// TIA Portal V17 export
// export: Created 2024-08-29T18:23:47.92153Z, ExportSetting WithDefaults, DisplayName Totally Integrated Automation Portal, DisplayVersion V17 Update 7, DisplayName TIA Portal Openness, DisplayVersion V17 Update 7, DisplayName TIA Portal Version Control Interface, DisplayVersion V17, DisplayName SINAMICS Startdrive Advanced, DisplayVersion V17 SP2, DisplayName SINAMICS Startdrive G110M, G120, G120C, G120D, G120P, G115D, DisplayVersion V17 SP2, DisplayName SINAMICS Startdrive G130, G150, S120, S150, SINAMICS MV, S210, DisplayVersion V17 SP2, DisplayName STEP 7 Professional, DisplayVersion V17 Update 7, DisplayName STEP 7 Safety, DisplayVersion V17 Update 6, DisplayName WinCC Advanced / Unified PC, DisplayVersion V17 Update 7
DATA_BLOCK "DB_SEND_IJCORE"   // DB1005
{ S7_Optimized_Access := 'FALSE' }
VERSION : 0.1
// stored: AutoNumber false, DBAccessibleFromOPCUA true, DBAccessibleFromWebserver true, IsOnlyStoredInLoadMemory false, IsWriteProtectedInAS false
   VAR
      Awake_DW : Word := 16#0000;
      Awake_SW : Int := 1;
      SW_Message : Array[1..300] of Word;
      Message : Array[1..50] of Struct
         Content : Array[1..80] of Byte;
      END_STRUCT;
   END_VAR
BEGIN
   SW_Message[1..8] := 16#FFFF;
   SW_Message[9..300] := 16#0000;
   Message[1].Content[1..80] := 16#00;
   Message[2].Content[1..80] := 16#00;
   Message[3].Content[1..80] := 16#00;
   Message[4].Content[1..80] := 16#00;
   Message[5].Content[1..80] := 16#00;
   Message[6].Content[1..80] := 16#00;
   Message[7].Content[1..80] := 16#00;
   Message[8].Content[1..80] := 16#00;
   Message[9].Content[1..80] := 16#00;
   Message[10].Content[1..80] := 16#00;
   Message[11].Content[1..80] := 16#00;
   Message[12].Content[1..80] := 16#00;
   Message[13].Content[1..80] := 16#00;
   Message[14].Content[1..80] := 16#00;
   Message[15].Content[1..80] := 16#00;
   Message[16].Content[1..80] := 16#00;
   Message[17].Content[1..80] := 16#00;
   Message[18].Content[1..80] := 16#00;
   Message[19].Content[1..80] := 16#00;
   Message[20].Content[1..80] := 16#00;
   Message[21].Content[1..80] := 16#00;
   Message[22].Content[1..80] := 16#00;
   Message[23].Content[1..80] := 16#00;
   Message[24].Content[1..80] := 16#00;
   Message[25].Content[1..80] := 16#00;
   Message[26].Content[1..80] := 16#00;
   Message[27].Content[1..80] := 16#00;
   Message[28].Content[1..80] := 16#00;
   Message[29].Content[1..80] := 16#00;
   Message[30].Content[1..80] := 16#00;
   Message[31].Content[1..80] := 16#00;
   Message[32].Content[1..80] := 16#00;
   Message[33].Content[1..80] := 16#00;
   Message[34].Content[1..80] := 16#00;
   Message[35].Content[1..80] := 16#00;
   Message[36].Content[1..80] := 16#00;
   Message[37].Content[1..80] := 16#00;
   Message[38].Content[1..80] := 16#00;
   Message[39].Content[1..80] := 16#00;
   Message[40].Content[1..80] := 16#00;
   Message[41].Content[1..80] := 16#00;
   Message[42].Content[1..80] := 16#00;
   Message[43].Content[1..80] := 16#00;
   Message[44].Content[1..80] := 16#00;
   Message[45].Content[1..80] := 16#00;
   Message[46].Content[1..80] := 16#00;
   Message[47].Content[1..80] := 16#00;
   Message[48].Content[1..80] := 16#00;
   Message[49].Content[1..80] := 16#00;
   Message[50].Content[1..80] := 16#00;
END_DATA_BLOCK
